# EPICS alarm handler configuration: mps_database/bareTest/alarms/areas/mpln_sph_mp04.alhConfig
GROUP NULL MPLN:SPH:MP04:1
$ALIAS MPS Link Node 123
$GUIDANCE
LTUH MPS
   Group Name: MPLN:SPH:MP04:1
   Summary PV:  MPLN:SPH:MP04:1:STATSUMY
$END
CHANNEL  MPLN:SPH:MP04:1    MPLN:SPH:MP04:1:MPS_EN_RBV		-----
CHANNEL  MPLN:SPH:MP04:1    MPLN:SPH:MP04:1:LC1_MODE_RBV		-----
